TYPE ST_SEQUENCE_PART :
STRUCT
	PARTID:DINT;
	STATUS:DINT;
	CURRENT_STEP:DINT;
	MESSAGE: STRING(100);
END_STRUCT
END_TYPE

(* stored: Version 1.1.0.1, ProductVersion 3.1.4024.15
   DUT ST_SEQUENCE_PART: Id {95e29eb6-c842-48bf-9a5b-2419e922b140} *)
